// Mitsubishi GX Works2 project: HMI 문자 표시하기 예시 코드   PLC: Q03UDV

PROGRAM MAIN
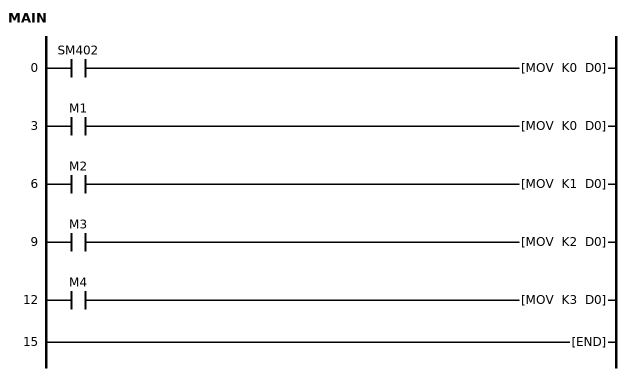
0     LD      SM402
      MOV     K0 D0
3     LD      M1
      MOV     K0 D0
6     LD      M2
      MOV     K1 D0
9     LD      M3
      MOV     K2 D0
12    LD      M4
      MOV     K3 D0
15    END
END_PROGRAM
